FUNCTION_BLOCK AgentFB (* Basic Function Block Type *)
  (* Standard: 61499-2 *)
  (* Version 0.2, 2003-12-04, JHC, Rockwell Automation, Renamed for better indexing. *)
  (* Version 0.1, 2002-11-05, JHC, Rockwell Automation, Corrected missing ST element in Algorithm REQ. *)
  (* Version 0.0, 2000-05-30, JHC, Rockwell Automation *)
  (* Compiler header: package fb.rt; *)
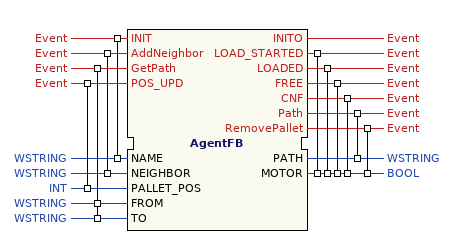
  EVENT_INPUT
    INIT WITH NAME; (* Initialization Request *)
    AddNeighbor WITH NEIGHBOR;
    GetPath WITH TO, FROM;
    POS_UPD WITH PALLET_POS;
  END_EVENT
  EVENT_OUTPUT
    INITO; (* Initialization Confirm *)
    LOAD_STARTED WITH MOTOR;
    LOADED WITH MOTOR;
    FREE WITH MOTOR;
    CNF WITH MOTOR;
    Path WITH PATH;
    RemovePallet WITH MOTOR;
  END_EVENT
  VAR_INPUT
    NAME : WSTRING;
    NEIGHBOR : WSTRING;
    PALLET_POS : INT;
    FROM : WSTRING;
    TO : WSTRING;
  END_VAR
  VAR_OUTPUT
    PATH : WSTRING;
    MOTOR : BOOL;
  END_VAR
END_FUNCTION_BLOCK
